Fanuc KAREL source: compact_preamble.KL

PROGRAM KT00438
%NOLOCKGROUP
VAR
I1:INTEGER;R2:REAL;OUT:BOOLEAN
BEGIN
I1=2
R2=3.0
OUT=((I1) >=R2)
END KT00438
